FUNCTION_BLOCK FB_FanControl_Test EXTENDS FB_TestSuite
VAR
END_VAR

METHOD FanSpeedMax
VAR
	FanControlRes: REAL;			//Actual value of FanControl
	ExpectedValue : REAL := 100;	//Expected value for FanControl

END_VAR
TEST('FanSpeedZero');
 
FanControlRes := FB_FanControl(fSpeed := 327.67);
 
AssertEquals(Expected := ExpectedValue,
             Actual := FanControlRes,
             Message := 'The calculation is not correct');
 
TEST_FINISHED();
END_METHOD

METHOD FanSpeedZero
VAR
	FanControlRes: REAL;		//Actual value of FanControl
	ExpectedValue : REAL := 0;	//Expected value for FanControl

END_VAR
TEST('FanSpeedZero');
 
FanControlRes := FB_FanControl(fSpeed := 0);
 
AssertEquals(Expected := ExpectedValue,
             Actual := FanControlRes,
             Message := 'The calculation is not correct');
 
TEST_FINISHED();
END_METHOD

END_FUNCTION_BLOCK

(* stored: Version 1.1.0.1, ProductVersion 3.1.4024.6
   POU FB_FanControl_Test: Id {25e59672-5b21-4b51-8765-679c25b545fe}, SpecialFunc None
   Method FanSpeedMax: Id {4dbabc29-d263-45c4-a9db-736404732271}
   Method FanSpeedZero: Id {909e3c1b-9eda-46c6-bea1-765e0c249ea9} *)
